FUNCTION_BLOCK ExistingAdapter (* Template for an empty basic function block *)
  (* Standard: 61499-2; Description: Copyright (c) 2019 Jan Holzweber This program and the accompanying materials are made available under the terms of the Eclipse Public License 2.0 which is available at https://www.eclipse.org/legal/epl-2.0/ SPDX-License-Identifier: EPL-2.0 *)
  (* Version 1.0, 2019-06-10, Jan Holzweber *)
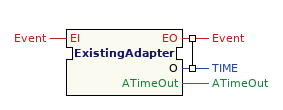
  EVENT_INPUT
    EI;
  END_EVENT
  EVENT_OUTPUT
    EO WITH O;
  END_EVENT
  VAR_OUTPUT
    O : TIME;
  END_VAR
  PLUGS
    ATimeOut : ATimeOut;
  END_PLUGS
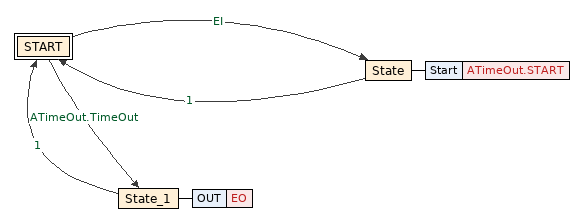
  EC_STATES
    START; (* Initial State *)
    State : Start -> ATimeOut.START;
    State_1 : OUT -> EO;
  END_STATES
  EC_TRANSITIONS
    START TO State := EI;
    State TO START := 1;
    START TO State_1 := ATimeOut.TimeOut;
    State_1 TO START := 1;
  END_TRANSITIONS
  ALGORITHM Start IN ST: (* new algorithm *)
ATimeOut.DT := T#10ms;
  END_ALGORITHM
  ALGORITHM OUT IN ST: (* new algorithm *)
O := ATimeOut.DT;
  END_ALGORITHM
END_FUNCTION_BLOCK
